{attribute 'qualified_only'}
VAR_GLOBAL
	
	rRefCylinderVel : REAL;
	rRefCylinderPos : REAL;
	rAutoTime : REAL;
	rCycleTime : REAL := 0.01;
	stStrokeRange : ST_pPistonStroke;
	rRunTime : REAL;
	rInitialStrokePosition : REAL;
END_VAR

(* stored: Version 1.1.0.1, ProductVersion 3.1.4024.10
   GVL parameter: Id {4f9916b1-2048-4311-979a-b33491aa40f3} *)
